FUNCTION_BLOCK Alarm
VAR_INPUT
	//Input that triggers the alarm condition
	Trigger : BOOL;
	//Alarm Acknowledge bit, Clears low priority alarms
	Alm_Ack : BOOL;
	//Alarm Reset, clears high priority alarms
	Reset : BOOL;
	//Alarm Priority, 1=Warning, 2=Error, 3=Critical
	Priority : INT;
	//Alarm Delay Setpoint in Seconds
	Delay_Setpoint : INT;
	//Alarm Enable
	Enable : BOOL;
END_VAR
VAR_OUTPUT
	//Alarm is triggered
	Active : BOOL;
END_VAR
VAR
	//Delay Timer Tags
	Delay_TON : TON;
	Delay_TON_PT : TIME;
	Delay_TON_ET : TIME;
	//Delay setpoint converted to Milliseconds
	Delay_mS : REAL;
	//Cutoff for needing to reset vs ack an alarm.  At or above this value requires reset.  
	Reset_Priority : REAL :=3;
END_VAR

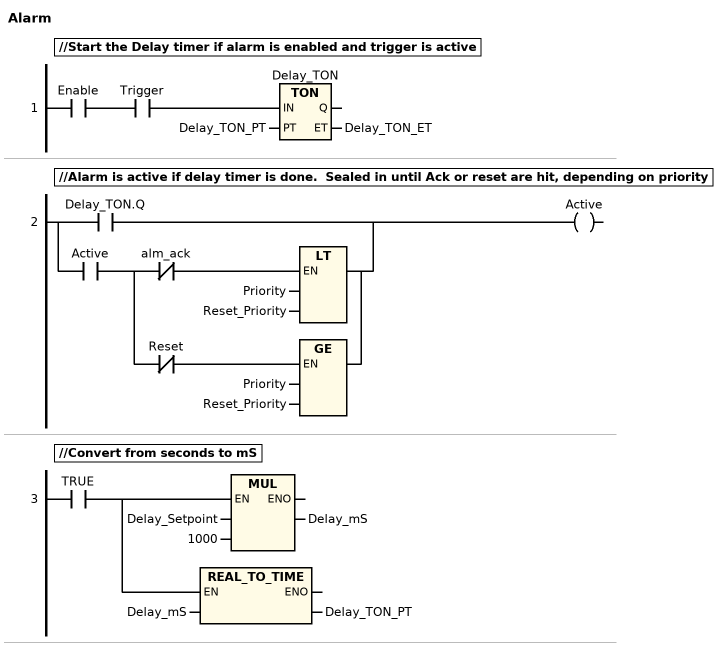
// NETWORK 1
// label: //Start the Delay timer if alarm is enabled and trigger is active
Delay_TON(IN := Enable AND Trigger, PT := Delay_TON_PT, ET => Delay_TON_ET); // TON

// NETWORK 2
// label: //Alarm is active if delay timer is done.  Sealed in until Ack or reset are hit, depending on priority
Active := Delay_TON.Q OR (Active AND NOT alm_ack AND Priority < Reset_Priority OR Active AND NOT Reset AND Priority >= Reset_Priority);

// NETWORK 3
// label: //Convert from seconds to mS
Delay_mS := Delay_Setpoint * 1000;
Delay_TON_PT := REAL_TO_TIME(Delay_mS);

END_FUNCTION_BLOCK

(* stored: Version 1.1.0.1, ProductVersion 3.1.4024.12
   POU Alarm: Id {4941c71f-2070-4068-8b1d-744b33ae24df}, SpecialFunc None *)
